// TIA Portal V20 export
DATA_BLOCK "SBK09"   // DB326
// stored: MemoryReserve 100
   VAR
      "SAFETY DOOR LOCK4.INPUT" : Bool := TRUE;
      "SAFETY DOOR LOCK5.INPUT" : Bool := TRUE;
      SPARE_5 : Bool := TRUE;
      SPARE : Bool := FALSE;
      "SAFETY DOOR LOCK4.INPUT_1" : Bool := FALSE;
      "SAFETY DOOR LOCK5.INPUT_1" : Bool := FALSE;
      SPARE_2 : Bool := FALSE;
      SPARE_3 : Bool := FALSE;
      "SAFETY DOOR LOCK4.OUTPUT" : Bool := FALSE;
      "SAFETY DOOR LOCK5.OUTPUT" : Bool := FALSE;
      SPARE_4 : Bool := FALSE;
   END_VAR
BEGIN
END_DATA_BLOCK
